// SIMATIC STEP 7 (V5.x) project RLI3_Profinet_400_300
// CPU: CPU 315-2 DP
// CPU: CPU 412-1
// station: Matériel
// station: SIMATIC 400(1)
// station: P_ADR_BUS
// station: Matériel
// station: SIMATIC 300(1)
// station: P_ADR_BUS
// program: Programme S7(1)
// program: Programme S7(2)

SYMBOL_TABLE
"GET"	SFB 14	SFB 14	// Read Data From a Remote CPU
"PUT"	SFB 15	SFB 15	// Write Data to a Remote CPU
"VAT_1"	VAT 1	
END_SYMBOL_TABLE

DATA_BLOCK DB 10
AUTHOR : SIMATIC
FAMILY : COM_FUNC
VERSION : 0.0
"PUT"
BEGIN
END_DATA_BLOCK

DATA_BLOCK DB 11
AUTHOR : SIMATIC
FAMILY : COM_FUNC
VERSION : 0.0
"PUT"
BEGIN
END_DATA_BLOCK

DATA_BLOCK DB 20
AUTHOR : SIMATIC
FAMILY : COM_FUNC
VERSION : 0.0
"GET"
BEGIN
END_DATA_BLOCK

ORGANIZATION_BLOCK OB 1
TITLE = "Main Program Sweep (Cycle)"
VERSION : 0.1
VAR_TEMP
  OB1_EV_CLASS : BYTE ;	//Bits 0-3 = 1 (Coming event), Bits 4-7 = 1 (Event class 1)
  OB1_SCAN_1 : BYTE ;	//1 (Cold restart scan 1 of OB 1), 3 (Scan 2-n of OB 1)
  OB1_PRIORITY : BYTE ;	//Priority of OB Execution
  OB1_OB_NUMBR : BYTE ;	//1 (Organization block 1, OB1)
  OB1_RESERVED_1 : BYTE ;	//Reserved for system
  OB1_RESERVED_2 : BYTE ;	//Reserved for system
  OB1_PREV_CYCLE : INT ;	//Cycle time of previous OB1 scan (milliseconds)
  OB1_MIN_CYCLE : INT ;	//Minimum cycle time of OB1 (milliseconds)
  OB1_MAX_CYCLE : INT ;	//Maximum cycle time of OB1 (milliseconds)
  OB1_DATE_TIME : DATE_AND_TIME ;	//Date and time OB1 started
END_VAR
BEGIN
NETWORK
TITLE =
NETWORK
TITLE =
      A     M 80.0;
      =     L 20.0;
      BLD   103;
      BLD   9;
      =     L 25.0;
      CDB;
      OPN   DI 11;
      TAR2  LD 21;
      A     L 20.0;
      =     DIX 0.0;
      L     1;
      T     DIW 2;
      L     W#16#1002;
      T     DIW 8;
      L     1;
      T     DIW 10;
      L     0;
      T     DIW 12;
      L     P#M 20.0;
      T     DID 14;
      L     W#16#1002;
      T     DIW 48;
      L     1;
      T     DIW 50;
      L     0;
      T     DIW 52;
      L     P#I 0.1;
      T     DID 54;
      LAR2  P#DBX 0.0;
      UC    "PUT";
      LAR2  LD 21;
      A     DIX 4.1;
      =     M 10.0;
      L     DIW 6;
      T     MW 15;
      CDB;
      BLD   10;
      NOP   0;
NETWORK
TITLE =
      A(;
      A     M 80.0;
      =     L 20.0;
      BLD   103;
      BLD   9;
      =     L 25.0;
      CDB;
      OPN   DI 20;
      TAR2  LD 21;
      A     L 20.0;
      =     DIX 0.0;
      L     1;
      T     DIW 2;
      L     W#16#1002;
      T     DIW 8;
      L     2;
      T     DIW 10;
      L     0;
      T     DIW 12;
      L     P#M 30.0;
      T     DID 14;
      L     W#16#1002;
      T     DIW 48;
      L     2;
      T     DIW 50;
      L     0;
      T     DIW 52;
      L     P#M 40.0;
      T     DID 54;
      LAR2  P#DBX 0.0;
      UC    "GET";
      LAR2  LD 21;
      A     DIX 4.1;
      =     M 2.0;
      L     DIW 6;
      T     MW 100;
      CDB;
      BLD   10;
      A     BR;
      );
      JNB   _001;
      L     MW 40;
      T     QW 0;
_001: NOP   0;
END_ORGANIZATION_BLOCK

SYMBOL_TABLE
"VAT_1"	VAT 1	
END_SYMBOL_TABLE

ORGANIZATION_BLOCK OB 1
TITLE = "Main Program Sweep (Cycle)"
VERSION : 0.1
VAR_TEMP
  OB1_EV_CLASS : BYTE ;	//Bits 0-3 = 1 (Coming event), Bits 4-7 = 1 (Event class 1)
  OB1_SCAN_1 : BYTE ;	//1 (Cold restart scan 1 of OB 1), 3 (Scan 2-n of OB 1)
  OB1_PRIORITY : BYTE ;	//Priority of OB Execution
  OB1_OB_NUMBR : BYTE ;	//1 (Organization block 1, OB1)
  OB1_RESERVED_1 : BYTE ;	//Reserved for system
  OB1_RESERVED_2 : BYTE ;	//Reserved for system
  OB1_PREV_CYCLE : INT ;	//Cycle time of previous OB1 scan (milliseconds)
  OB1_MIN_CYCLE : INT ;	//Minimum cycle time of OB1 (milliseconds)
  OB1_MAX_CYCLE : INT ;	//Maximum cycle time of OB1 (milliseconds)
  OB1_DATE_TIME : DATE_AND_TIME ;	//Date and time OB1 started
END_VAR
BEGIN
NETWORK
TITLE =
      A     M 20.1;
      CU    C 10;
      A     M 20.2;
      CD    C 10;
      NOP   0;
      NOP   0;
      A     I 0.7;
      R     C 10;
      NOP   0;
      LC    C 10;
      T     MW 30;
      NOP   0;
END_ORGANIZATION_BLOCK
